FUNCTION_BLOCK DIV_INT (* IEC 61131-3 INT Division *)
  (* Standard: 61131-3 *)
  (* Version 0.0, 2004-12-15, JHC, Rockwell Automation, Converted from SRC format. *)
  (* Compiler header: package fb.rt.plc.math; *)
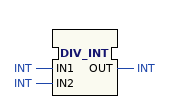
  VAR_INPUT
    IN1 : INT; (* Dividend *)
    IN2 : INT; (* Divisor *)
  END_VAR
  VAR_OUTPUT
    OUT : INT; (* Quotient *)
  END_VAR
END_FUNCTION_BLOCK
